Staubli VAL3: VAL3help_example.pjx

--- VAL3help_example.pjx ---
Parameters version=s8.3Cs9_BS845 stackSize=5000 millimeterUnit=true
Program file=exit.pgx
Program file=start.pgx
Program file=stop.pgx
Data file=VAL3help_example.dtx

--- VAL3help_example.dtx ---
mdesc mNomSpeed
string sInput
string sOutput
string sPrompt
num nRet
bool bExit

--- start.pgx ---
program start()
begin
  // Init variables
  sPrompt="Please enter your input:"
  sInput=""
  sOutput=""
  bExit = false

  // Display user page
  nRet=userPage("main")

  if (userPagePrompt(sPrompt, sInput) == true)
    // TODO:
    // Add hereafter your code with sInput as input and sOutput as output
    // For example sOutput=sInput
     sOutput=sInput
  else
    sOutput="User canceled prompt"
  endIf

  // Wait for button exit to be pressed
  while bExit==false
    delay(0)
  endWhile
end

--- exit.pgx ---
program exit()
begin
  bExit = true
end
